FUNCTION_BLOCK PumpController
VAR
	volumePump					: VolumePump;
	eState						: ( DISABLED, ENABLED, PUMPING, PUMPING_COMPLETE );
	requestButton				: I_Button;
	juiceSetter					: Potentiometer;
	ledDisplay					: AnalogLedDisplay010;
	fJuiceSetpointInMililiters	: LREAL;
	fMinSetRangeInMililiters	: LREAL;
	fMaxSetRangeInMililiters	: LREAL;
END_VAR

volumePump();

CASE eState OF
	
	DISABLED:
		;
		
	ENABLED:
		ledDisplay.SetValue(juiceSetter.ActualValue);
		IF requestButton.IsPressed THEN
			fJuiceSetpointInMililiters := F_Scale ( juiceSetter.ActualValue, 0, 32767, fMinSetRangeInMililiters, fMaxSetRangeInMililiters );
			eState := PUMPING;
		END_IF
		
	PUMPING:
		ledDisplay.SetValue( TO_INT (F_Scale ( fJuiceSetpointInMililiters - volumePump.PumpedJuiceInMililiters, fMinSetRangeInMililiters, fMaxSetRangeInMililiters, 0, 32767 ) ) );
		volumePump.Start();
		IF volumePump.PumpedJuiceInMililiters >= fJuiceSetpointInMililiters THEN
			volumePump.Reset();
			eState := PUMPING_COMPLETE;
		END_IF
		
	PUMPING_COMPLETE:
		;
		
END_CASE

METHOD Disable : BOOL
VAR_INPUT
END_VAR
eState := DISABLED;
END_METHOD

METHOD Enable : BOOL
VAR_INPUT
END_VAR
eState := ENABLED;
END_METHOD

//FB_Init is always available implicitly and it is used primarily for initialization.
//The return value is not evaluated. For a specific influence, you can also declare the
//methods explicitly and provide additional code there with the standard initialization
//code. You can evaluate the return value.
METHOD FB_Init: BOOL
VAR_INPUT
    bInitRetains: BOOL; // TRUE: the retain variables are initialized (reset warm / reset cold)
    bInCopyCode: BOOL;  // TRUE: the instance will be copied to the copy code afterward (online change)   
	requestButton				: I_Button;
	fMinSetRangeInMililiters	: LREAL;
	fMaxSetRangeInMililiters	: LREAL;
END_VAR
THIS^.requestButton := requestButton;
THIS^.fMinSetRangeInMililiters := LIMIT(0, fMinSetRangeInMililiters, 10_000);
THIS^.fMaxSetRangeInMililiters := LIMIT(0, fMaxSetRangeInMililiters, 10_000);
END_METHOD

PROPERTY IsDisabled : BOOL
GET
IsDisabled := eState = DISABLED;
END_GET
END_PROPERTY

PROPERTY IsEnabled : BOOL
GET
IsEnabled := eState = ENABLED;
END_GET
END_PROPERTY

PROPERTY IsPumping : BOOL
GET
IsPumping := eState = PUMPING;
END_GET
END_PROPERTY

PROPERTY IsPumpingComplete : BOOL
GET
IsPumpingComplete := eState = PUMPING_COMPLETE;
END_GET
END_PROPERTY

END_FUNCTION_BLOCK

(* stored: Version 1.1.0.1
   POU PumpController: Id {c47f4e83-f94f-490b-a79c-636f640ba23b}, SpecialFunc None
   Method Disable: Id {1e3c5ceb-0153-4b8c-9ea3-700faacaa6ac}
   Method Enable: Id {497b6319-3591-4ae7-80ca-b5ce422abe5c}
   Method FB_Init: Id {fa7fc71d-e7e3-4466-99fc-835ddc8d2f31}
   Property IsDisabled: Id {1865061b-bc09-4052-85d3-935e08fd9a37}
   Get Get: Id {25809d9d-b7bd-4ab9-a65b-492e51fdc7f2}
   Property IsEnabled: Id {b6d963a5-7c14-466e-bbcb-f2652bc1da7c}
   Get Get: Id {71a3abb8-4628-4e75-b1c4-a868e3e355fb}
   Property IsPumping: Id {a312785a-3bbf-4f14-b0a9-fdcb2e5e66ca}
   Get Get: Id {fab194c9-7642-47b3-87ef-57bf3c21532b}
   Property IsPumpingComplete: Id {4ad76a02-0bcf-46e9-b2e3-02f9b0513c61}
   Get Get: Id {31f9fd02-8a2e-4e49-8361-b87a3d69366c} *)
